FUNCTION_BLOCK Testowy
VAR
END_VAR

END_FUNCTION_BLOCK

(* stored: Version 1.1.0.1
   POU Testowy: Id {70677787-d308-4bbe-8726-95dea33bce6a}, SpecialFunc None *)
